// TIA Portal project "Motor_StartStop_V2" (V18)

(* hardware
DEVICE "S7-1200 station_1"  S7-1200 Station
   slot 0: "Rack_0"  S7-1200 Rack  Rack  V1.0
   slot 1: "PLC_1"  CPU 1214C DC/DC/DC  6ES7 214-1AG40-0XB0  V4.6
*)

// ===== PLC "PLC_1"  CPU 1214C DC/DC/DC =====

VAR_GLOBAL   // PLC tag table "Default tag table"
   "Start_button" AT %I0.0 : Bool;
   "Stop_button" AT %I0.1 : Bool;
   "Motor_Output" AT %Q0.0 : Bool;
END_VAR

ORGANIZATION_BLOCK "Main"   // OB1, LAD, ProgramCycle
TITLE = "Main Program Sweep (Cycle)"
{ S7_Optimized_Access := 'TRUE' }
VERSION : 0.1
   VAR_INPUT
      Initial_Call : Bool;   // Initial call of this OB
      Remanence : Bool;   // =True, if remanent data are available
   END_VAR
BEGIN

REGION Network 1
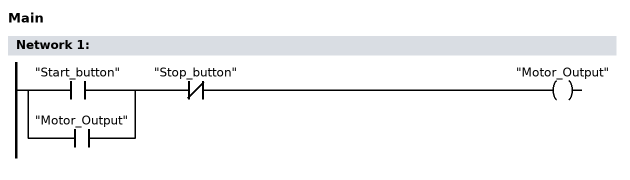
   RUNG wire#powerrail
      Contact( "Start_button" )
      wire#w1
      I_Contact( "Stop_button" )
      Coil( "Motor_Output" )
   END_RUNG
   RUNG wire#powerrail
      Contact( "Motor_Output" )
   END_RUNG wire#w1
   // the same network as SCL:
   "Motor_Output" := ("Start_button" OR "Motor_Output") AND NOT "Stop_button";
END_REGION
END_ORGANIZATION_BLOCK